SUBAPPLICATION NumericValue_PHYS_TO_NVS (* Numerischer VT-Wert (PHYS-Variante, skaliert) einlesen und in NVS speichern (generisch). *)
  (* Standard: 61499-2 *)
  (* Version 1.0, 2026-09-09, Franz Höpfinger, Meisterschulen am Ostbahnhof, Ausgelagert aus Uebung_012f_sub zur Wiederverwendung. *)
  PACKAGE MyLib::sys;
  IMPORT isobus::UT::Q::const::IDs::ID_NULL;
  IMPORT logiBUS::utils::conversion::phys::NumericObjectPool_S;
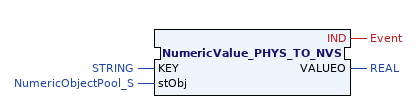
  EVENT_OUTPUT
    IND;
  END_EVENT
  VAR_INPUT
    KEY : STRING; (* Key name. *)
    stObj : logiBUS::utils::conversion::phys::NumericObjectPool_S := (u16ObjId := ID_NULL, r32Scale := 1.0, i32Offset := 0, u8Decimals := 0);
  END_VAR
  VAR_OUTPUT
    VALUEO : REAL;
  END_VAR
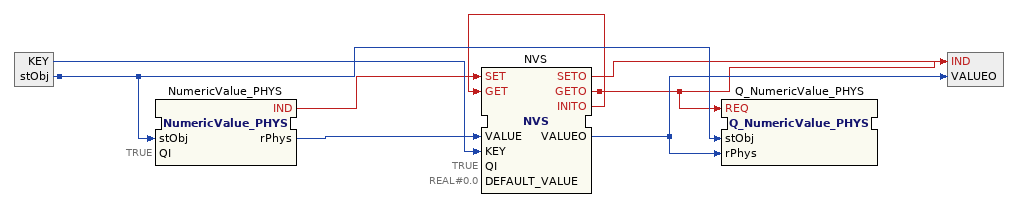
  FBS
    NumericValue_PHYS : isobus::UT::io::NumericValue::NumericValue_PHYS(QI := TRUE);
    NVS : logiBUS::storage::esp32_nvs::NVS(QI := TRUE, DEFAULT_VALUE := REAL#0.0);
    Q_NumericValue_PHYS : isobus::UT::Q::Q_NumericValue_PHYS;
  END_FBS
  EVENT_CONNECTIONS
    NumericValue_PHYS.IND TO NVS.SET;
    NVS.SETO TO IND;
    NVS.GETO TO Q_NumericValue_PHYS.REQ;
    NVS.GETO TO IND;
    NVS.INITO TO NVS.GET;
  END_CONNECTIONS
  DATA_CONNECTIONS
    NumericValue_PHYS.rPhys TO NVS.VALUE;
    stObj TO Q_NumericValue_PHYS.stObj;
    KEY TO NVS.KEY;
    NVS.VALUEO TO Q_NumericValue_PHYS.rPhys;
    NVS.VALUEO TO VALUEO;
    stObj TO NumericValue_PHYS.stObj;
  END_CONNECTIONS
END_SUBAPPLICATION
